FUNCTION_BLOCK Master (* Basic Function Block Type *)
  (* Standard: 61499-2 *)
  (* Version 0.0, 1/14/2024, midxav, Template *)
  PACKAGE Main;
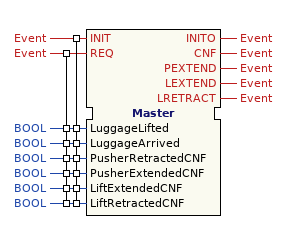
  EVENT_INPUT
    INIT WITH LuggageLifted, LuggageArrived, PusherRetractedCNF, LiftRetractedCNF, LiftExtendedCNF, PusherExtendedCNF; (* Initialization Request *)
    REQ WITH LuggageLifted, LuggageArrived, PusherRetractedCNF, LiftRetractedCNF, LiftExtendedCNF, PusherExtendedCNF; (* Normal Execution Request *)
  END_EVENT
  EVENT_OUTPUT
    INITO; (* Initialization Confirm *)
    CNF; (* Execution Confirmation *)
    PEXTEND;
    LEXTEND;
    LRETRACT;
  END_EVENT
  VAR_INPUT
    LuggageLifted : BOOL;
    LuggageArrived : BOOL;
    PusherRetractedCNF : BOOL;
    PusherExtendedCNF : BOOL;
    LiftExtendedCNF : BOOL;
    LiftRetractedCNF : BOOL;
  END_VAR
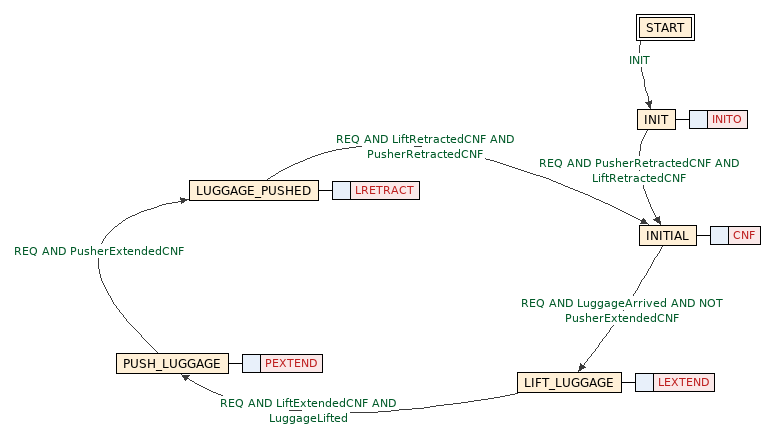
  EC_STATES
    START; (* Initial State *)
    INIT : -> INITO; (* Initialization *)
    INITIAL : -> CNF;
    LIFT_LUGGAGE : -> LEXTEND;
    PUSH_LUGGAGE : -> PEXTEND;
    LUGGAGE_PUSHED : -> LRETRACT;
  END_STATES
  EC_TRANSITIONS
    START TO INIT := INIT;
    INIT TO INITIAL := REQ AND PusherRetractedCNF AND LiftRetractedCNF;
    INITIAL TO LIFT_LUGGAGE := REQ AND LuggageArrived AND NOT PusherExtendedCNF;
    LIFT_LUGGAGE TO PUSH_LUGGAGE := REQ AND LiftExtendedCNF AND LuggageLifted;
    PUSH_LUGGAGE TO LUGGAGE_PUSHED := REQ AND PusherExtendedCNF;
    LUGGAGE_PUSHED TO INITIAL := REQ AND LiftRetractedCNF AND PusherRetractedCNF;
  END_TRANSITIONS
END_FUNCTION_BLOCK
